// TIA Portal V17 export
// export: Created 2022-07-31T06:40:45.0685756Z, ExportSetting WithDefaults, DisplayName Totally Integrated Automation Portal, DisplayVersion V17 Update 2, DisplayName TIA Portal Openness, DisplayVersion V17 Update 2, DisplayName TIA Portal Version Control Interface, DisplayVersion V17, DisplayName SINAMICS Startdrive Advanced, DisplayVersion V17 Update1, DisplayName SINAMICS Startdrive G110M, G120, G120C, G120D, G120P, G115D, DisplayVersion V17 Update1, DisplayName SINAMICS Startdrive G130, G150, S120, S150, SINAMICS MV, S210, DisplayVersion V17 Update1, DisplayName STEP 7 Professional, DisplayVersion V17 Update 2, DisplayName STEP 7 Safety, DisplayVersion V17, DisplayName WinCC UA Professional, DisplayVersion V17 Update 2
DATA_BLOCK "LoggerLevels"   // DB3
{ S7_Optimized_Access := 'TRUE'; DB_Accessible_From_OPC_UA := 'FALSE' }
VERSION : 0.1
// stored: AutoNumber true, DBAccessibleFromOPCUA false, DBAccessibleFromWebserver false, IsOnlyStoredInLoadMemory false, IsRetainMemResEnabled false, IsWriteProtectedInAS false, MemoryReserve 100
   VAR
      NOTSET { ExternalAccessible := 'False'; ExternalVisible := 'False'; ExternalWritable := 'False'} : USInt := 0;   // logging everything
      DEBUG { ExternalAccessible := 'False'; ExternalVisible := 'False'; ExternalWritable := 'False'} : USInt := 10;
      INFO { ExternalAccessible := 'False'; ExternalVisible := 'False'; ExternalWritable := 'False'} : USInt := 20;
      WARNING { ExternalAccessible := 'False'; ExternalVisible := 'False'; ExternalWritable := 'False'} : USInt := 30;
      ERROR { ExternalAccessible := 'False'; ExternalVisible := 'False'; ExternalWritable := 'False'} : USInt := 40;
      CRITICAL { ExternalAccessible := 'False'; ExternalVisible := 'False'; ExternalWritable := 'False'} : USInt := 50;
      DISABLE { ExternalAccessible := 'False'; ExternalVisible := 'False'; ExternalWritable := 'False'} : USInt := 100;   // logging disabled
   END_VAR
BEGIN
END_DATA_BLOCK
